FUNCTION_BLOCK XBAR_CTL (* Transfer Bar Control *)
  (* Standard: 61499-1; Classification: Simulation; ApplicationDomain: Material Handling; Function: Control; Type: Transfer Bar *)
  (* Version 0.0, 2002-05-20, JHC, Rockwell Automation *)
  (* Compiler header: package fb.rt.mach; *)
  (* Compiler Java IBM Jikes 1.06 *)
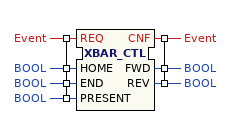
  EVENT_INPUT
    REQ WITH HOME, END, PRESENT;
  END_EVENT
  EVENT_OUTPUT
    CNF WITH FWD, REV;
  END_EVENT
  VAR_INPUT
    HOME : BOOL; (* Bar at HOME position *)
    END : BOOL; (* Bar at END position *)
    PRESENT : BOOL; (* Workpiece Present *)
  END_VAR
  VAR_OUTPUT
    FWD : BOOL; (* Drive Forward *)
    REV : BOOL; (* Drive Backward *)
  END_VAR
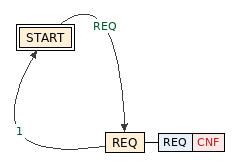
  EC_STATES
    START;
    REQ : REQ -> CNF;
  END_STATES
  EC_TRANSITIONS
    START TO REQ := REQ;
    REQ TO START := 1;
  END_TRANSITIONS
  ALGORITHM REQ IN LD:
    FWD := END ! PRESENT & ;
    REV := HOME ! PRESENT ! & ;
  END_ALGORITHM
END_FUNCTION_BLOCK
